PROGRAM PRG_CASE_ValidateContentManual
VAR
	fbCase_ValidateContent		: FB_CASE_ValidateContent;
	
	
	(* Init function/method declarations*)
	rTrigDataInit		: R_TRIG;
	bDataInit			: BOOL;
	iOuter				: INT;
	iPack				: INT;
	sPackNum			: STRING;
	sOuterNum			: STRING;
	sPackCode			: STRING;
	
	(* Inputs *)
	bExecute 					: BOOL;
	stCTDateTime				: ST_SYSTEM_DateTime;	(* CaseTrace date/time structure *)
	
	(* In/Out *)
	stProductInstruction		: ST_PCM_Status;
	nSecquentionalCounter		: UDINT;
	stCodeInfo_Outer			: ST_CodeInfo;
	stCaseRejectReasons			: ST_RejectReasonsForCase;
	stCACData 					: ST_CAC_Data;
	
	(* Outputs *)
	bDone 						: BOOL;
	bBusy						: BOOL;
	bError						: BOOL;
	nErrorID 					: UDINT;

	sRejectCode					: T_MaxString;
	nValidationIndex			: INT;
	
END_VAR

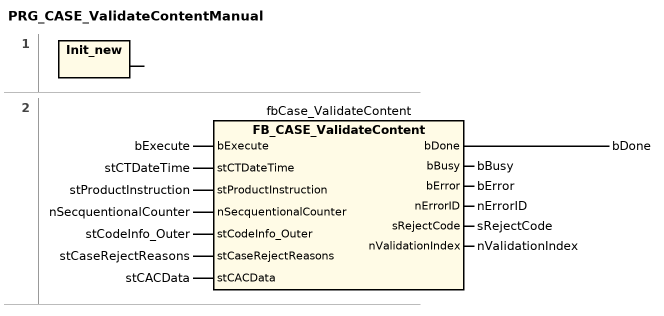
// NETWORK 1
Init_new();

// NETWORK 2
fbCase_ValidateContent(
    bExecute := bExecute,
    stCTDateTime := stCTDateTime,
    stProductInstruction := stProductInstruction,
    nSecquentionalCounter := nSecquentionalCounter,
    stCodeInfo_Outer := stCodeInfo_Outer,
    stCaseRejectReasons := stCaseRejectReasons,
    stCACData := stCACData,
    bBusy => bBusy,
    bError => bError,
    nErrorID => nErrorID,
    sRejectCode => sRejectCode,
    nValidationIndex => nValidationIndex); // FB_CASE_ValidateContent
bDone := fbCase_ValidateContent.bDone;

ACTION Init:
rTrigDataInit(CLK := bDataInit);

IF rTrigDataInit.Q THEN
		
	stProductInstruction.nOutersPerCase		:= 50;
	stProductInstruction.nPacksPerOuter 	:= 10;











	FOR iOuter := 1 TO stProductInstruction.nOutersPerCase DO
		(* Ustaw outer *)
		stCACData.Outer[iOuter].Barcode    := CONCAT('OUTER', INT_TO_STRING(iOuter));
		stCACData.Outer[iOuter].OuterCodeStatus := 5;
		






		FOR iPack := 1 TO stProductInstruction.nPacksPerOuter DO
			(* Pack number z zerami *)
			sPackNum := CONCAT('0', INT_TO_STRING(iPack));  (* dla 1-9: '01'-'09' *)
			IF iPack = 10 THEN
				sPackNum := '10';
			END_IF;
			
			(* Outer number z zerami dla 1-9 *)
			sOuterNum := CONCAT('0', INT_TO_STRING(iOuter));
			IF iOuter >= 10 THEN
				sOuterNum := INT_TO_STRING(iOuter);
			END_IF;
			
			(* Sklej pack code *)
			sPackCode := CONCAT(CONCAT('PACK', sPackNum), CONCAT('OUTER', sOuterNum));
			
			(* Przypisz *)
			stCACData.Outer[iOuter].PackCode[iPack]			:= sPackCode;
			stCACData.Outer[iOuter].PackCodeStatus[iPack]	:= 5;
			stCACData.Outer[iOuter].PackRejectID[iPack]		:= 0;


			
		END_FOR;
	END_FOR;	










	
END_IF
END_ACTION

ACTION Init_new:

rTrigDataInit(CLK := bDataInit);

IF rTrigDataInit.Q THEN
	
	MEMSET(ADR(stCACData), 16#00, SIZEOF(stCACData));	
	
	stProductInstruction.nOutersPerCase 	:= 50;
	stProductInstruction.nPacksPerOuter		:= 10;	
	// jezeli tej wartosci nie ma, jest na 0 i czytaj ponizej
	stProductInstruction.nPacksPerCase		:= 500;
	stProductInstruction.nOpMode			:= 11;
	stProductInstruction.sRetailSKU			:= '1234567';
	stProductInstruction.nAcceptanceLevel 	:= 10;

	// jezeli stCACData.NumberOfOuters=0 , czyli usune te linie ponizej to nie wejdzie do warunku linia 40 FB_CASE_ValidateContent i wywali
	// jakis error z elsifa ktoregos
	stCACData.NumberOfOuters			:= stProductInstruction.nOutersPerCase;
	stCACData.CodingAndTrackingMode		:= stProductInstruction.nOpMode;
	stCACData.RetailSKU					:= stProductInstruction.sRetailSKU;

	FOR iOuter := 1 TO stProductInstruction.nOutersPerCase DO
		(* Outer number z zerami *)
		sOuterNum := F_StringAddPrefix(INT_TO_STRING(iOuter),2,'0');
	
		stCACData.Outer[iOuter].Barcode    				:= CONCAT('OUTER', sOuterNum);
		stCACData.Outer[iOuter].NumberOfPacks 			:= stProductInstruction.nPacksPerOuter;
		stCACData.Outer[iOuter].NumberOfLinkedPacks 	:= stProductInstruction.nPacksPerOuter;
		stCACData.Outer[iOuter].AcceptanceLevel 		:= stProductInstruction.nAcceptanceLevel;
		stCACData.Outer[iOuter].CodingAndTrackingMode	:= stProductInstruction.nOpMode;
		stCACData.Outer[iOuter].OuterRejectCode			:= 'OK';
	
		FOR iPack := 1 TO stProductInstruction.nPacksPerOuter DO
			(* Pack number dwucyfrowy z zerami *)
			sPackNum := F_StringAddPrefix(INT_TO_STRING(iPack),2,'0');			
			(* Sklej pack code *)
			sPackCode := CONCAT(CONCAT('PACK', sPackNum), CONCAT('OUTER', sOuterNum));
			
			(* Write Pack Barcodes / Data*)
			stCACData.Outer[iOuter].PackCode[iPack]				:= sPackCode;
			stCACData.Outer[iOuter].PackCodeStatus[iPack]		:= 5;
			stCACData.Outer[iOuter].PackRejectID[iPack]			:= 0;			
			stCACData.Outer[iOuter].PackRejectCode[iPack]		:= 'OK';			
			stCACData.Outer[iOuter].PackCodeStatus[iPack].5 	:= TRUE;
			
			
			IF iPack = 1 THEN
				stCACData.Outer[iOuter].AggregationCodes[1]	:= stCACData.Outer[iOuter].PackCode[iPack];
			END_IF
			IF iPack = 2 THEN
				stCACData.Outer[iOuter].AggregationCodes[2]	:= stCACData.Outer[iOuter].PackCode[iPack];
			END_IF
		END_FOR
	END_FOR	
	
	stCACData.Outer[3].OuterCodeStatus.5 	:= TRUE;
	stCACData.Outer[4].OuterCodeStatus.5	:= TRUE;
	
	stCACData.NumberOfOuters 				:= 55;
	
END_IF
END_ACTION

END_PROGRAM

(* stored: Version 1.1.0.1
   POU PRG_CASE_ValidateContentManual: Id {4b02fdb6-ccf7-458c-96cb-c09b4d69eaf2}, SpecialFunc None
   Action Init: Id {a36de12f-b054-405c-a8cb-ac1230cd4e58}
   Action Init_new: Id {907ed0a9-63d3-498c-b872-2e22bfbcd3c4} *)
